FUNCTION_BLOCK PUBLIC DATE_TO_TestSuite EXTENDS TcUnit.FB_TestSuite
VAR
END_VAR

Check_DATE_TO_BOOL_Max();
Check_DATE_TO_BOOL_Min();
Check_DATE_TO_BYTE_Max();
Check_DATE_TO_BYTE_Min();
Check_DATE_TO_BYTE_TooHigh();
Check_DATE_TO_WORD_Max();
Check_DATE_TO_WORD_Min();
Check_DATE_TO_WORD_TooHigh();
Check_DATE_TO_DWORD_Max();
Check_DATE_TO_DWORD_Min();
Check_DATE_TO_LWORD_Max();
Check_DATE_TO_LWORD_Min();
Check_DATE_TO_SINT_Max();
Check_DATE_TO_SINT_Min();
Check_DATE_TO_SINT_TooHigh();
Check_DATE_TO_INT_Max();
Check_DATE_TO_INT_Min();
Check_DATE_TO_INT_TooHigh();
Check_DATE_TO_DINT_Max();
Check_DATE_TO_DINT_Min();
Check_DATE_TO_DINT_TooHigh();
Check_DATE_TO_LINT_Max();
Check_DATE_TO_LINT_Min();
Check_DATE_TO_USINT_Max();
Check_DATE_TO_USINT_Min();
Check_DATE_TO_USINT_TooHigh();
Check_DATE_TO_UINT_Max();
Check_DATE_TO_UINT_Min();
Check_DATE_TO_UINT_TooHigh();
Check_DATE_TO_UDINT_Max();
Check_DATE_TO_UDINT_Min();
Check_DATE_TO_ULINT_Max();
Check_DATE_TO_ULINT_Min();
Check_DATE_TO_REAL_Max();
Check_DATE_TO_REAL_Min();
Check_DATE_TO_LREAL_Max();
Check_DATE_TO_LREAL_Min();
Check_DATE_TO_TIME_Max();
Check_DATE_TO_TIME_Min();
Check_DATE_TO_TIME_TooHigh();
Check_DATE_TO_TOD_Max();
Check_DATE_TO_TOD_Min();
Check_DATE_TO_TOD_TooHigh();
Check_DATE_TO_DATE_Max();
Check_DATE_TO_DATE_Min();
Check_DATE_TO_DT_Max();
Check_DATE_TO_DT_Min();
Check_DATE_TO_STRING_Max();
Check_DATE_TO_STRING_Min();

METHOD PUBLIC Check_DATE_TO_BOOL_Min
VAR
	value : DATE := DatatypeLimits.DATE_MIN_VALUE;
	actual : BOOL;
	converted : BOOL;
	equal : BOOL;
END_VAR
TEST('Check_DATE_TO_BOOL_Min');

// @TEST-RUN
converted := TryConvert_DATE_TO_Destination(value, actual);
equal := actual = DATE_TO_BOOL(value);

// @TEST-ASSERT
AssertTrue(Condition := equal, Message := 'Did not convert DATE to BOOL correctly');
AssertTrue(Condition := converted, Message := 'Did not report DATE to BOOL conversion was successful');

TEST_FINISHED();
END_METHOD

METHOD PUBLIC Check_DATE_TO_BOOL_Max
VAR
	value : DATE := DatatypeLimits.DATE_MAX_VALUE;
	actual : BOOL;
	converted : BOOL;
	equal : BOOL;
END_VAR
TEST('Check_DATE_TO_BOOL_Max');

// @TEST-RUN
converted := TryConvert_DATE_TO_Destination(value, actual);
equal := actual = DATE_TO_BOOL(value);

// @TEST-ASSERT
AssertTrue(Condition := equal, Message := 'Did not convert DATE to BOOL correctly');
AssertTrue(Condition := converted, Message := 'Did not report DATE to BOOL conversion was successful');

TEST_FINISHED();
END_METHOD

METHOD PUBLIC Check_DATE_TO_BYTE_Min
VAR
	value : DATE := DatatypeLimits.DATE_MIN_VALUE;
	actual : BYTE;
	converted : BOOL;
	equal : BOOL;
END_VAR
TEST('Check_DATE_TO_BYTE_Min');

// @TEST-RUN
converted := TryConvert_DATE_TO_Destination(value, actual);
equal := actual = DATE_TO_BYTE(value);

// @TEST-ASSERT
AssertTrue(Condition := equal, Message := 'Did not convert DATE to BYTE correctly');
AssertTrue(Condition := converted, Message := 'Did not report DATE to BYTE conversion was successful');

TEST_FINISHED();
END_METHOD

METHOD PUBLIC Check_DATE_TO_BYTE_TooHigh
VAR
	value : DATE := DatatypeLimits.DATE_MAX_VALUE;
	actual : BYTE;
	converted : BOOL;
END_VAR
TEST('Check_DATE_TO_BYTE_TooHigh');

// @TEST-RUN
converted := TryConvert_DATE_TO_Destination(value, actual);

// @TEST-ASSERT
AssertFalse(Condition := converted, Message := 'Did not report DATE to BYTE conversion was prevented');

TEST_FINISHED();
END_METHOD

METHOD PUBLIC Check_DATE_TO_BYTE_Max
VAR
	value : DATE := DatatypeLimits.MAX_VALUE_OF_DATE_WHICH_CAN_BE_HELD_IN_A_BYTE;
	actual : BYTE;
	converted : BOOL;
	equal : BOOL;
END_VAR
TEST('Check_DATE_TO_BYTE_Max');

// @TEST-RUN
converted := TryConvert_DATE_TO_Destination(value, actual);
equal := actual = DATE_TO_BYTE(value);

// @TEST-ASSERT
AssertTrue(Condition := equal, Message := 'Did not convert DATE to BYTE correctly');
AssertTrue(Condition := converted, Message := 'Did not report DATE to BYTE conversion was successful');

TEST_FINISHED();
END_METHOD

METHOD PUBLIC Check_DATE_TO_DATE_Min
VAR
	value : DATE := DatatypeLimits.DATE_MIN_VALUE;
	actual : DATE;
	converted : BOOL;
	equal : BOOL;
END_VAR
TEST('Check_DATE_TO_DATE_Min');

// @TEST-RUN
converted := TryConvert_DATE_TO_Destination(value, actual);
equal := actual = value;

// @TEST-ASSERT
AssertTrue(Condition := equal, Message := 'Did not convert DATE to DATE correctly');
AssertTrue(Condition := converted, Message := 'Did not report DATE to DATE conversion was successful');

TEST_FINISHED();
END_METHOD

METHOD PUBLIC Check_DATE_TO_DATE_Max
VAR
	value : DATE := DatatypeLimits.DATE_MAX_VALUE;
	actual : DATE;
	converted : BOOL;
	equal : BOOL;
END_VAR
TEST('Check_DATE_TO_DATE_Max');

// @TEST-RUN
converted := TryConvert_DATE_TO_Destination(value, actual);
equal := actual = value;

// @TEST-ASSERT
AssertTrue(Condition := equal, Message := 'Did not convert DATE to DATE correctly');
AssertTrue(Condition := converted, Message := 'Did not report DATE to DATE conversion was successful');

TEST_FINISHED();
END_METHOD

METHOD PUBLIC Check_DATE_TO_DINT_Min
VAR
	value : DATE := DatatypeLimits.DATE_MIN_VALUE;
	actual : DINT;
	converted : BOOL;
	equal : BOOL;
END_VAR
TEST('Check_DATE_TO_DINT_Min');

// @TEST-RUN
converted := TryConvert_DATE_TO_Destination(value, actual);
equal := actual = DATE_TO_DINT(value);

// @TEST-ASSERT
AssertTrue(Condition := equal, Message := 'Did not convert DATE to DINT correctly');
AssertTrue(Condition := converted, Message := 'Did not report DATE to DINT conversion was successful');

TEST_FINISHED();
END_METHOD

METHOD PUBLIC Check_DATE_TO_DINT_TooHigh
VAR
	value : DATE := DatatypeLimits.DATE_MAX_VALUE;
	actual : DINT;
	converted : BOOL;
END_VAR
TEST('Check_DATE_TO_DINT_TooHigh');

// @TEST-RUN
converted := TryConvert_DATE_TO_Destination(value, actual);

// @TEST-ASSERT
AssertFalse(Condition := converted, Message := 'Did not report DATE to DINT conversion was prevented');

TEST_FINISHED();
END_METHOD

METHOD PUBLIC Check_DATE_TO_DINT_Max
VAR
	value : DATE := DatatypeLimits.MAX_VALUE_OF_DATE_WHICH_CAN_BE_HELD_IN_A_DINT;
	actual : DINT;
	converted : BOOL;
	equal : BOOL;
END_VAR
TEST('Check_DATE_TO_DINT_Max');

// @TEST-RUN
converted := TryConvert_DATE_TO_Destination(value, actual);
equal := actual = DATE_TO_DINT(value);

// @TEST-ASSERT
AssertTrue(Condition := equal, Message := 'Did not convert DATE to DINT correctly');
AssertTrue(Condition := converted, Message := 'Did not report DATE to DINT conversion was successful');

TEST_FINISHED();
END_METHOD

METHOD PUBLIC Check_DATE_TO_DT_Min
VAR
	value : DATE := DatatypeLimits.DATE_MIN_VALUE;
	actual : DT;
	converted : BOOL;
	equal : BOOL;
END_VAR
TEST('Check_DATE_TO_DT_Min');

// @TEST-RUN
converted := TryConvert_DATE_TO_Destination(value, actual);
equal := actual = DATE_TO_DT(value);

// @TEST-ASSERT
AssertTrue(Condition := equal, Message := 'Did not convert DATE to DT correctly');
AssertTrue(Condition := converted, Message := 'Did not report DATE to DT conversion was successful');

TEST_FINISHED();
END_METHOD

METHOD PUBLIC Check_DATE_TO_DT_Max
VAR
	value : DATE := DatatypeLimits.MAX_VALUE_OF_DATE_WHICH_CAN_BE_HELD_IN_A_DT;
	actual : DT;
	converted : BOOL;
	equal : BOOL;
END_VAR
TEST('Check_DATE_TO_DT_Max');

// @TEST-RUN
converted := TryConvert_DATE_TO_Destination(value, actual);
equal := actual = DATE_TO_DT(value);

// @TEST-ASSERT
AssertTrue(Condition := equal, Message := 'Did not convert DATE to DT correctly');
AssertTrue(Condition := converted, Message := 'Did not report DATE to DT conversion was successful');

TEST_FINISHED();
END_METHOD

METHOD PUBLIC Check_DATE_TO_DWORD_Min
VAR
	value : DATE := DatatypeLimits.DATE_MIN_VALUE;
	actual : DWORD;
	converted : BOOL;
	equal : BOOL;
END_VAR
TEST('Check_DATE_TO_DWORD_Min');

// @TEST-RUN
converted := TryConvert_DATE_TO_Destination(value, actual);
equal := actual = DATE_TO_DWORD(value);

// @TEST-ASSERT
AssertTrue(Condition := equal, Message := 'Did not convert DATE to DWORD correctly');
AssertTrue(Condition := converted, Message := 'Did not report DATE to DWORD conversion was successful');

TEST_FINISHED();
END_METHOD

METHOD PUBLIC Check_DATE_TO_DWORD_Max
VAR
	value : DATE := DatatypeLimits.DATE_MAX_VALUE;
	actual : DWORD;
	converted : BOOL;
	equal : BOOL;
END_VAR
TEST('Check_DATE_TO_DWORD_Max');

// @TEST-RUN
converted := TryConvert_DATE_TO_Destination(value, actual);
equal := actual = DATE_TO_DWORD(value);

// @TEST-ASSERT
AssertTrue(Condition := equal, Message := 'Did not convert DATE to DWORD correctly');
AssertTrue(Condition := converted, Message := 'Did not report DATE to DWORD conversion was successful');

TEST_FINISHED();
END_METHOD

METHOD PUBLIC Check_DATE_TO_INT_Min
VAR
	value : DATE := DatatypeLimits.DATE_MIN_VALUE;
	actual : INT;
	converted : BOOL;
	equal : BOOL;
END_VAR
TEST('Check_DATE_TO_INT_Min');

// @TEST-RUN
converted := TryConvert_DATE_TO_Destination(value, actual);
equal := actual = DATE_TO_INT(value);

// @TEST-ASSERT
AssertTrue(Condition := equal, Message := 'Did not convert DATE to INT correctly');
AssertTrue(Condition := converted, Message := 'Did not report DATE to INT conversion was successful');

TEST_FINISHED();
END_METHOD

METHOD PUBLIC Check_DATE_TO_INT_TooHigh
VAR
	value : DATE := DatatypeLimits.DATE_MAX_VALUE;
	actual : INT;
	converted : BOOL;
END_VAR
TEST('Check_DATE_TO_INT_TooHigh');

// @TEST-RUN
converted := TryConvert_DATE_TO_Destination(value, actual);

// @TEST-ASSERT
AssertFalse(Condition := converted, Message := 'Did not report DATE to INT conversion was prevented');

TEST_FINISHED();
END_METHOD

METHOD PUBLIC Check_DATE_TO_INT_Max
VAR
	value : DATE := DatatypeLimits.MAX_VALUE_OF_DATE_WHICH_CAN_BE_HELD_IN_A_INT;
	actual : INT;
	converted : BOOL;
	equal : BOOL;
END_VAR
TEST('Check_DATE_TO_INT_Max');

// @TEST-RUN
converted := TryConvert_DATE_TO_Destination(value, actual);
equal := actual = DATE_TO_INT(value);

// @TEST-ASSERT
AssertTrue(Condition := equal, Message := 'Did not convert DATE to INT correctly');
AssertTrue(Condition := converted, Message := 'Did not report DATE to INT conversion was successful');

TEST_FINISHED();
END_METHOD

METHOD PUBLIC Check_DATE_TO_LINT_Min
VAR
	value : DATE := DatatypeLimits.DATE_MIN_VALUE;
	actual : LINT;
	converted : BOOL;
	equal : BOOL;
END_VAR
TEST('Check_DATE_TO_LINT_Min');

// @TEST-RUN
converted := TryConvert_DATE_TO_Destination(value, actual);
equal := actual = DATE_TO_LINT(value);

// @TEST-ASSERT
AssertTrue(Condition := equal, Message := 'Did not convert DATE to LINT correctly');
AssertTrue(Condition := converted, Message := 'Did not report DATE to LINT conversion was successful');

TEST_FINISHED();
END_METHOD

METHOD PUBLIC Check_DATE_TO_LINT_Max
VAR
	value : DATE := DatatypeLimits.DATE_MAX_VALUE;
	actual : LINT;
	converted : BOOL;
	equal : BOOL;
END_VAR
TEST('Check_DATE_TO_LINT_Max');

// @TEST-RUN
converted := TryConvert_DATE_TO_Destination(value, actual);
equal := actual = DATE_TO_LINT(value);

// @TEST-ASSERT
AssertTrue(Condition := equal, Message := 'Did not convert DATE to LINT correctly');
AssertTrue(Condition := converted, Message := 'Did not report DATE to LINT conversion was successful');

TEST_FINISHED();
END_METHOD

METHOD PUBLIC Check_DATE_TO_LREAL_Min
VAR
	value : DATE := DatatypeLimits.DATE_MIN_VALUE;
	actual : LREAL;
	converted : BOOL;
	equal : BOOL;
END_VAR
TEST('Check_DATE_TO_LREAL_Min');

// @TEST-RUN
converted := TryConvert_DATE_TO_Destination(value, actual);
equal := actual = DATE_TO_LREAL(value);

// @TEST-ASSERT
AssertTrue(Condition := equal, Message := 'Did not convert DATE to LREAL correctly');
AssertTrue(Condition := converted, Message := 'Did not report DATE to LREAL conversion was successful');

TEST_FINISHED();
END_METHOD

METHOD PUBLIC Check_DATE_TO_LREAL_Max
VAR
	value : DATE := DatatypeLimits.DATE_MAX_VALUE;
	actual : LREAL;
	converted : BOOL;
	equal : BOOL;
END_VAR
TEST('Check_DATE_TO_LREAL_Max');

// @TEST-RUN
converted := TryConvert_DATE_TO_Destination(value, actual);
equal := actual = DATE_TO_LREAL(value);

// @TEST-ASSERT
AssertTrue(Condition := equal, Message := 'Did not convert DATE to LREAL correctly');
AssertTrue(Condition := converted, Message := 'Did not report DATE to LREAL conversion was successful');

TEST_FINISHED();
END_METHOD

METHOD PUBLIC Check_DATE_TO_LWORD_Min
VAR
	value : DATE := DatatypeLimits.DATE_MIN_VALUE;
	actual : LWORD;
	converted : BOOL;
	equal : BOOL;
END_VAR
TEST('Check_DATE_TO_LWORD_Min');

// @TEST-RUN
converted := TryConvert_DATE_TO_Destination(value, actual);
equal := actual = DATE_TO_LWORD(value);

// @TEST-ASSERT
AssertTrue(Condition := equal, Message := 'Did not convert DATE to LWORD correctly');
AssertTrue(Condition := converted, Message := 'Did not report DATE to LWORD conversion was successful');

TEST_FINISHED();
END_METHOD

METHOD PUBLIC Check_DATE_TO_LWORD_Max
VAR
	value : DATE := DatatypeLimits.DATE_MAX_VALUE;
	actual : LWORD;
	converted : BOOL;
	equal : BOOL;
END_VAR
TEST('Check_DATE_TO_LWORD_Max');

// @TEST-RUN
converted := TryConvert_DATE_TO_Destination(value, actual);
equal := actual = DATE_TO_LWORD(value);

// @TEST-ASSERT
AssertTrue(Condition := equal, Message := 'Did not convert DATE to LWORD correctly');
AssertTrue(Condition := converted, Message := 'Did not report DATE to LWORD conversion was successful');

TEST_FINISHED();
END_METHOD

METHOD PUBLIC Check_DATE_TO_REAL_Min
VAR
	value : DATE := DatatypeLimits.DATE_MIN_VALUE;
	actual : REAL;
	converted : BOOL;
	equal : BOOL;
END_VAR
TEST('Check_DATE_TO_REAL_Min');

// @TEST-RUN
converted := TryConvert_DATE_TO_Destination(value, actual);
equal := actual = DATE_TO_REAL(value);

// @TEST-ASSERT
AssertTrue(Condition := equal, Message := 'Did not convert DATE to REAL correctly');
AssertTrue(Condition := converted, Message := 'Did not report DATE to REAL conversion was successful');

TEST_FINISHED();
END_METHOD

METHOD PUBLIC Check_DATE_TO_REAL_Max
VAR
	value : DATE := DatatypeLimits.DATE_MAX_VALUE;
	actual : REAL;
	converted : BOOL;
	equal : BOOL;
END_VAR
TEST('Check_DATE_TO_REAL_Max');

// @TEST-RUN
converted := TryConvert_DATE_TO_Destination(value, actual);
equal := actual = DATE_TO_REAL(value);

// @TEST-ASSERT
AssertTrue(Condition := equal, Message := 'Did not convert DATE to REAL correctly');
AssertTrue(Condition := converted, Message := 'Did not report DATE to REAL conversion was successful');

TEST_FINISHED();
END_METHOD

METHOD PUBLIC Check_DATE_TO_SINT_Min
VAR
	value : DATE := DatatypeLimits.DATE_MIN_VALUE;
	actual : SINT;
	converted : BOOL;
	equal : BOOL;
END_VAR
TEST('Check_DATE_TO_SINT_Min');

// @TEST-RUN
converted := TryConvert_DATE_TO_Destination(value, actual);
equal := actual = DATE_TO_SINT(value);

// @TEST-ASSERT
AssertTrue(Condition := equal, Message := 'Did not convert DATE to SINT correctly');
AssertTrue(Condition := converted, Message := 'Did not report DATE to SINT conversion was successful');

TEST_FINISHED();
END_METHOD

METHOD PUBLIC Check_DATE_TO_SINT_TooHigh
VAR
	value : DATE := DatatypeLimits.DATE_MAX_VALUE;
	actual : SINT;
	converted : BOOL;
END_VAR
TEST('Check_DATE_TO_SINT_TooHigh');

// @TEST-RUN
converted := TryConvert_DATE_TO_Destination(value, actual);

// @TEST-ASSERT
AssertFalse(Condition := converted, Message := 'Did not report DATE to SINT conversion was prevented');

TEST_FINISHED();
END_METHOD

METHOD PUBLIC Check_DATE_TO_SINT_Max
VAR
	value : DATE := DatatypeLimits.MAX_VALUE_OF_DATE_WHICH_CAN_BE_HELD_IN_A_SINT;
	actual : SINT;
	converted : BOOL;
	equal : BOOL;
END_VAR
TEST('Check_DATE_TO_SINT_Max');

// @TEST-RUN
converted := TryConvert_DATE_TO_Destination(value, actual);
equal := actual = DATE_TO_SINT(value);

// @TEST-ASSERT
AssertTrue(Condition := equal, Message := 'Did not convert DATE to SINT correctly');
AssertTrue(Condition := converted, Message := 'Did not report DATE to SINT conversion was successful');

TEST_FINISHED();
END_METHOD

METHOD PUBLIC Check_DATE_TO_STRING_Min
VAR
	value : DATE := DatatypeLimits.DATE_MIN_VALUE;
	actual : STRING;
	converted : BOOL;
	equal : BOOL;
END_VAR
TEST('Check_DATE_TO_STRING_Min');

// @TEST-RUN
converted := TryConvert_DATE_TO_Destination(value, actual);
equal := actual = DATE_TO_STRING(value);

// @TEST-ASSERT
AssertTrue(Condition := equal, Message := 'Did not convert DATE to STRING correctly');
AssertTrue(Condition := converted, Message := 'Did not report DATE to STRING conversion was successful');

TEST_FINISHED();
END_METHOD

METHOD PUBLIC Check_DATE_TO_STRING_Max
VAR
	value : DATE := DatatypeLimits.DATE_MAX_VALUE;
	actual : STRING;
	converted : BOOL;
	equal : BOOL;
END_VAR
TEST('Check_DATE_TO_STRING_Max');

// @TEST-RUN
converted := TryConvert_DATE_TO_Destination(value, actual);
equal := actual = DATE_TO_STRING(value);

// @TEST-ASSERT
AssertTrue(Condition := equal, Message := 'Did not convert DATE to STRING correctly');
AssertTrue(Condition := converted, Message := 'Did not report DATE to STRING conversion was successful');

TEST_FINISHED();
END_METHOD

METHOD PUBLIC Check_DATE_TO_TIME_Min
VAR
	value : DATE := DatatypeLimits.DATE_MIN_VALUE;
	actual : TIME;
	converted : BOOL;
	equal : BOOL;
END_VAR
TEST('Check_DATE_TO_TIME_Min');

// @TEST-RUN
converted := TryConvert_DATE_TO_Destination(value, actual);
equal := actual = DATE_TO_TIME(value);

// @TEST-ASSERT
AssertTrue(Condition := equal, Message := 'Did not convert DATE to TIME correctly');
AssertTrue(Condition := converted, Message := 'Did not report DATE to TIME conversion was successful');

TEST_FINISHED();
END_METHOD

METHOD PUBLIC Check_DATE_TO_TIME_TooHigh
VAR
	value : DATE := DatatypeLimits.DATE_MAX_VALUE;
	actual : TIME;
	converted : BOOL;
END_VAR
TEST('Check_DATE_TO_TIME_TooHigh');

// @TEST-RUN
converted := TryConvert_DATE_TO_Destination(value, actual);

// @TEST-ASSERT
AssertFalse(Condition := converted, Message := 'Did not report DATE to TIME conversion was prevented');

TEST_FINISHED();
END_METHOD

METHOD PUBLIC Check_DATE_TO_TIME_Max
VAR
	value : DATE := DatatypeLimits.MAX_VALUE_OF_DATE_WHICH_CAN_BE_HELD_IN_A_TIME;
	actual : TIME;
	converted : BOOL;
	equal : BOOL;
END_VAR
TEST('Check_DATE_TO_TIME_Max');

// @TEST-RUN
converted := TryConvert_DATE_TO_Destination(value, actual);
equal := actual = DATE_TO_TIME(value);

// @TEST-ASSERT
AssertTrue(Condition := equal, Message := 'Did not convert DATE to TIME correctly');
AssertTrue(Condition := converted, Message := 'Did not report DATE to TIME conversion was successful');

TEST_FINISHED();
END_METHOD

METHOD PUBLIC Check_DATE_TO_TOD_Min
VAR
	value : DATE := DatatypeLimits.DATE_MIN_VALUE;
	actual : TOD;
	converted : BOOL;
	equal : BOOL;
END_VAR
TEST('Check_DATE_TO_TOD_Min');

// @TEST-RUN
converted := TryConvert_DATE_TO_Destination(value, actual);
equal := actual = DATE_TO_TOD(value);

// @TEST-ASSERT
AssertTrue(Condition := equal, Message := 'Did not convert DATE to TOD correctly');
AssertTrue(Condition := converted, Message := 'Did not report DATE to TOD conversion was successful');

TEST_FINISHED();
END_METHOD

METHOD PUBLIC Check_DATE_TO_TOD_TooHigh
VAR
	value : DATE := DatatypeLimits.DATE_MAX_VALUE;
	actual : TOD;
	converted : BOOL;
END_VAR
TEST('Check_DATE_TO_TOD_TooHigh');

// @TEST-RUN
converted := TryConvert_DATE_TO_Destination(value, actual);

// @TEST-ASSERT
AssertFalse(Condition := converted, Message := 'Did not report DATE to TOD conversion was prevented');

TEST_FINISHED();
END_METHOD

METHOD PUBLIC Check_DATE_TO_TOD_Max
VAR
	value : DATE := DatatypeLimits.MAX_VALUE_OF_DATE_WHICH_CAN_BE_HELD_IN_A_TOD;
	actual : TOD;
	converted : BOOL;
	equal : BOOL;
END_VAR
TEST('Check_DATE_TO_TOD_Max');

// @TEST-RUN
converted := TryConvert_DATE_TO_Destination(value, actual);
equal := actual = DATE_TO_TOD(value);

// @TEST-ASSERT
AssertTrue(Condition := equal, Message := 'Did not convert DATE to TOD correctly');
AssertTrue(Condition := converted, Message := 'Did not report DATE to TOD conversion was successful');

TEST_FINISHED();
END_METHOD

METHOD PUBLIC Check_DATE_TO_UDINT_Min
VAR
	value : DATE := DatatypeLimits.DATE_MIN_VALUE;
	actual : UDINT;
	converted : BOOL;
	equal : BOOL;
END_VAR
TEST('Check_DATE_TO_UDINT_Min');

// @TEST-RUN
converted := TryConvert_DATE_TO_Destination(value, actual);
equal := actual = DATE_TO_UDINT(value);

// @TEST-ASSERT
AssertTrue(Condition := equal, Message := 'Did not convert DATE to UDINT correctly');
AssertTrue(Condition := converted, Message := 'Did not report DATE to UDINT conversion was successful');

TEST_FINISHED();
END_METHOD

METHOD PUBLIC Check_DATE_TO_UDINT_Max
VAR
	value : DATE := DatatypeLimits.DATE_MAX_VALUE;
	actual : UDINT;
	converted : BOOL;
	equal : BOOL;
END_VAR
TEST('Check_DATE_TO_UDINT_Max');

// @TEST-RUN
converted := TryConvert_DATE_TO_Destination(value, actual);
equal := actual = DATE_TO_UDINT(value);

// @TEST-ASSERT
AssertTrue(Condition := equal, Message := 'Did not convert DATE to UDINT correctly');
AssertTrue(Condition := converted, Message := 'Did not report DATE to UDINT conversion was successful');

TEST_FINISHED();
END_METHOD

METHOD PUBLIC Check_DATE_TO_UINT_Min
VAR
	value : DATE := DatatypeLimits.DATE_MIN_VALUE;
	actual : UINT;
	converted : BOOL;
	equal : BOOL;
END_VAR
TEST('Check_DATE_TO_UINT_Min');

// @TEST-RUN
converted := TryConvert_DATE_TO_Destination(value, actual);
equal := actual = DATE_TO_UINT(value);

// @TEST-ASSERT
AssertTrue(Condition := equal, Message := 'Did not convert DATE to UINT correctly');
AssertTrue(Condition := converted, Message := 'Did not report DATE to UINT conversion was successful');

TEST_FINISHED();
END_METHOD

METHOD PUBLIC Check_DATE_TO_UINT_TooHigh
VAR
	value : DATE := DatatypeLimits.DATE_MAX_VALUE;
	actual : UINT;
	converted : BOOL;
END_VAR
TEST('Check_DATE_TO_UINT_TooHigh');

// @TEST-RUN
converted := TryConvert_DATE_TO_Destination(value, actual);

// @TEST-ASSERT
AssertFalse(Condition := converted, Message := 'Did not report DATE to UINT conversion was prevented');

TEST_FINISHED();
END_METHOD

METHOD PUBLIC Check_DATE_TO_UINT_Max
VAR
	value : DATE := DatatypeLimits.MAX_VALUE_OF_DATE_WHICH_CAN_BE_HELD_IN_A_UINT;
	actual : UINT;
	converted : BOOL;
	equal : BOOL;
END_VAR
TEST('Check_DATE_TO_UINT_Max');

// @TEST-RUN
converted := TryConvert_DATE_TO_Destination(value, actual);
equal := actual = DATE_TO_UINT(value);

// @TEST-ASSERT
AssertTrue(Condition := equal, Message := 'Did not convert DATE to UINT correctly');
AssertTrue(Condition := converted, Message := 'Did not report DATE to UINT conversion was successful');

TEST_FINISHED();
END_METHOD

METHOD PUBLIC Check_DATE_TO_ULINT_Min
VAR
	value : DATE := DatatypeLimits.DATE_MIN_VALUE;
	actual : ULINT;
	converted : BOOL;
	equal : BOOL;
END_VAR
TEST('Check_DATE_TO_ULINT_Min');

// @TEST-RUN
converted := TryConvert_DATE_TO_Destination(value, actual);
equal := actual = DATE_TO_ULINT(value);

// @TEST-ASSERT
AssertTrue(Condition := equal, Message := 'Did not convert DATE to ULINT correctly');
AssertTrue(Condition := converted, Message := 'Did not report DATE to ULINT conversion was successful');

TEST_FINISHED();
END_METHOD

METHOD PUBLIC Check_DATE_TO_ULINT_Max
VAR
	value : DATE := DatatypeLimits.DATE_MAX_VALUE;
	actual : ULINT;
	converted : BOOL;
	equal : BOOL;
END_VAR
TEST('Check_DATE_TO_ULINT_Max');

// @TEST-RUN
converted := TryConvert_DATE_TO_Destination(value, actual);
equal := actual = DATE_TO_ULINT(value);

// @TEST-ASSERT
AssertTrue(Condition := equal, Message := 'Did not convert DATE to ULINT correctly');
AssertTrue(Condition := converted, Message := 'Did not report DATE to ULINT conversion was successful');

TEST_FINISHED();
END_METHOD

METHOD PUBLIC Check_DATE_TO_USINT_Min
VAR
	value : DATE := DatatypeLimits.DATE_MIN_VALUE;
	actual : USINT;
	converted : BOOL;
	equal : BOOL;
END_VAR
TEST('Check_DATE_TO_USINT_Min');

// @TEST-RUN
converted := TryConvert_DATE_TO_Destination(value, actual);
equal := actual = DATE_TO_USINT(value);

// @TEST-ASSERT
AssertTrue(Condition := equal, Message := 'Did not convert DATE to USINT correctly');
AssertTrue(Condition := converted, Message := 'Did not report DATE to USINT conversion was successful');

TEST_FINISHED();
END_METHOD

METHOD PUBLIC Check_DATE_TO_USINT_TooHigh
VAR
	value : DATE := DatatypeLimits.DATE_MAX_VALUE;
	actual : USINT;
	converted : BOOL;
END_VAR
TEST('Check_DATE_TO_USINT_TooHigh');

// @TEST-RUN
converted := TryConvert_DATE_TO_Destination(value, actual);

// @TEST-ASSERT
AssertFalse(Condition := converted, Message := 'Did not report DATE to USINT conversion was prevented');

TEST_FINISHED();
END_METHOD

METHOD PUBLIC Check_DATE_TO_USINT_Max
VAR
	value : DATE := DatatypeLimits.MAX_VALUE_OF_DATE_WHICH_CAN_BE_HELD_IN_A_USINT;
	actual : USINT;
	converted : BOOL;
	equal : BOOL;
END_VAR
TEST('Check_DATE_TO_USINT_Max');

// @TEST-RUN
converted := TryConvert_DATE_TO_Destination(value, actual);
equal := actual = DATE_TO_USINT(value);

// @TEST-ASSERT
AssertTrue(Condition := equal, Message := 'Did not convert DATE to USINT correctly');
AssertTrue(Condition := converted, Message := 'Did not report DATE to USINT conversion was successful');

TEST_FINISHED();
END_METHOD

METHOD PUBLIC Check_DATE_TO_WORD_Min
VAR
	value : DATE := DatatypeLimits.DATE_MIN_VALUE;
	actual : WORD;
	converted : BOOL;
	equal : BOOL;
END_VAR
TEST('Check_DATE_TO_WORD_Min');

// @TEST-RUN
converted := TryConvert_DATE_TO_Destination(value, actual);
equal := actual = DATE_TO_WORD(value);

// @TEST-ASSERT
AssertTrue(Condition := equal, Message := 'Did not convert DATE to WORD correctly');
AssertTrue(Condition := converted, Message := 'Did not report DATE to WORD conversion was successful');

TEST_FINISHED();
END_METHOD

METHOD PUBLIC Check_DATE_TO_WORD_TooHigh
VAR
	value : DATE := DatatypeLimits.DATE_MAX_VALUE;
	actual : WORD;
	converted : BOOL;
END_VAR
TEST('Check_DATE_TO_WORD_TooHigh');

// @TEST-RUN
converted := TryConvert_DATE_TO_Destination(value, actual);

// @TEST-ASSERT
AssertFalse(Condition := converted, Message := 'Did not report DATE to WORD conversion was prevented');

TEST_FINISHED();
END_METHOD

METHOD PUBLIC Check_DATE_TO_WORD_Max
VAR
	value : DATE := DatatypeLimits.MAX_VALUE_OF_DATE_WHICH_CAN_BE_HELD_IN_A_WORD;
	actual : WORD;
	converted : BOOL;
	equal : BOOL;
END_VAR
TEST('Check_DATE_TO_WORD_Max');

// @TEST-RUN
converted := TryConvert_DATE_TO_Destination(value, actual);
equal := actual = DATE_TO_WORD(value);

// @TEST-ASSERT
AssertTrue(Condition := equal, Message := 'Did not convert DATE to WORD correctly');
AssertTrue(Condition := converted, Message := 'Did not report DATE to WORD conversion was successful');

TEST_FINISHED();
END_METHOD

END_FUNCTION_BLOCK

(* stored: Version 1.1.0.1, ProductVersion 3.1.4024.12
   POU DATE_TO_TestSuite: Id {55bde9b3-96c0-48a1-8e64-4fcacc2d6d2f}, SpecialFunc None
   Method Check_DATE_TO_BOOL_Min: Id {2d447892-0a6d-4d61-ba89-203c05f50f7e}
   Method Check_DATE_TO_BOOL_Max: Id {8190d19d-6da8-455e-a66b-581b8d873acc}
   Method Check_DATE_TO_BYTE_Min: Id {cba1714c-ecb1-41f6-9834-782d2df40fc9}
   Method Check_DATE_TO_BYTE_TooHigh: Id {ae00b03e-2bc4-4a33-881d-cbead2193bba}
   Method Check_DATE_TO_BYTE_Max: Id {cdf81856-1a62-46c3-9e59-224d7670a3c6}
   Method Check_DATE_TO_DATE_Min: Id {4416668d-03a8-4ed3-a5b0-20eef169d746}
   Method Check_DATE_TO_DATE_Max: Id {b6893444-e169-4ae4-9288-740844db7f68}
   Method Check_DATE_TO_DINT_Min: Id {a6a5844e-6d65-44d6-a1e6-2b9fd15aa826}
   Method Check_DATE_TO_DINT_TooHigh: Id {9f20fe60-f5ab-461a-b595-cbf85bd197e8}
   Method Check_DATE_TO_DINT_Max: Id {6ce5bf3d-981e-4d2d-95b8-d0e8e0c8d585}
   Method Check_DATE_TO_DT_Min: Id {aa0135ae-8ba1-42cc-9388-4c9a2fd46ea6}
   Method Check_DATE_TO_DT_Max: Id {a16f076d-2c1b-4144-a3a9-e4bd5af84faa}
   Method Check_DATE_TO_DWORD_Min: Id {72d5b52a-5045-4463-a71f-ca5a81ac6a24}
   Method Check_DATE_TO_DWORD_Max: Id {45645ba6-fe12-420c-ae3e-9a4a28c626bd}
   Method Check_DATE_TO_INT_Min: Id {2b999bf5-3893-4678-b24a-361b0992688b}
   Method Check_DATE_TO_INT_TooHigh: Id {ce4abbfa-4b36-4a3b-a81e-e035393d524e}
   Method Check_DATE_TO_INT_Max: Id {48f7f351-eacc-48ee-b2a1-3113dbd00b7c}
   Method Check_DATE_TO_LINT_Min: Id {fe3846ba-905e-47a5-bd2e-cda673207d0f}
   Method Check_DATE_TO_LINT_Max: Id {8d7fd2d3-ee56-4518-bb30-59841f1d7535}
   Method Check_DATE_TO_LREAL_Min: Id {536af5b5-9599-47fa-a45a-f1db4974709e}
   Method Check_DATE_TO_LREAL_Max: Id {172f471b-fad8-4749-a9ba-d42e1d079ecc}
   Method Check_DATE_TO_LWORD_Min: Id {1bdb8492-6b03-42b8-b943-ec814883db0c}
   Method Check_DATE_TO_LWORD_Max: Id {9457f517-886a-43ec-a9e9-888de3dc784e}
   Method Check_DATE_TO_REAL_Min: Id {a97486ba-d3f4-400a-857e-1836a26c0d23}
   Method Check_DATE_TO_REAL_Max: Id {43205fc5-7b2f-4673-8bce-7c26154df23e}
   Method Check_DATE_TO_SINT_Min: Id {be299111-2f3f-406b-a5e1-c2ecc5c11f82}
   Method Check_DATE_TO_SINT_TooHigh: Id {cfe8bb14-7c80-4d59-af8c-9b73758d553f}
   Method Check_DATE_TO_SINT_Max: Id {2c9a267b-2514-46b6-9aec-c8fb8d9099b9}
   Method Check_DATE_TO_STRING_Min: Id {c3185aaf-28aa-4489-a6ff-9197327c22ca}
   Method Check_DATE_TO_STRING_Max: Id {5fb99f8c-cebf-4f7f-a578-262cde4f75f5}
   Method Check_DATE_TO_TIME_Min: Id {0b57a8b3-861e-45da-99d0-cff806bc0b5a}
   Method Check_DATE_TO_TIME_TooHigh: Id {c49c3ba3-b5ea-409e-bf09-c4cac657a3bc}
   Method Check_DATE_TO_TIME_Max: Id {d8d1a71d-5755-4332-8bb8-5c62445be712}
   Method Check_DATE_TO_TOD_Min: Id {c8e374ba-1a22-4b1f-b9ff-0cb7ee99c566}
   Method Check_DATE_TO_TOD_TooHigh: Id {fd748e69-9735-4bfc-8a7d-482e283a6fa7}
   Method Check_DATE_TO_TOD_Max: Id {cd4673e6-5114-4192-8656-7edf8e49be6d}
   Method Check_DATE_TO_UDINT_Min: Id {6f8b5438-f32a-4c8a-a378-4695314e9eb4}
   Method Check_DATE_TO_UDINT_Max: Id {1012ca3b-96bd-41a2-902b-e4818f75e5ab}
   Method Check_DATE_TO_UINT_Min: Id {46fa3800-f640-4b9f-bfb7-f8e5fa02801d}
   Method Check_DATE_TO_UINT_TooHigh: Id {69f3118e-f697-4493-a059-ec215b1d0cfe}
   Method Check_DATE_TO_UINT_Max: Id {afbcb556-af46-4282-a635-968b21baffe7}
   Method Check_DATE_TO_ULINT_Min: Id {f60f61f9-6c72-4f32-bc96-3efbdea1a798}
   Method Check_DATE_TO_ULINT_Max: Id {89810b30-a8f3-4315-b68a-73c13f5897d1}
   Method Check_DATE_TO_USINT_Min: Id {fbda16f4-0bfd-43b0-ae3e-7cf9c87f3df4}
   Method Check_DATE_TO_USINT_TooHigh: Id {f3b55807-cb7e-4d42-b371-864d1b39dd95}
   Method Check_DATE_TO_USINT_Max: Id {32524afa-d702-4436-9217-23bcb783e198}
   Method Check_DATE_TO_WORD_Min: Id {879db07e-30a6-4ba9-b8dc-e77ceb23d03d}
   Method Check_DATE_TO_WORD_TooHigh: Id {f9fc827d-bf9f-4f18-bb9e-0a352de6f9b8}
   Method Check_DATE_TO_WORD_Max: Id {de6c2978-2123-4c12-a437-961de3522928} *)
